{attribute 'GeneratedUsingTerminal: EL6752--0000'}
{attribute addProperty BoxType "EL6752--0000"}
{attribute addProperty Id "InfoDataAT %I*InfoData_90184F0C16"}
{attribute addProperty CRC "554310285"}
{attribute addProperty Size "16"}
TYPE EL6752_210A1A8D EXTENDS EtcSlaveTerminalBase_947E5A46 :
STRUCT
	{attribute addProperty Name "InfoData"}
	InfoData : InfoData_90184F0C;
END_STRUCT
END_TYPE

(* stored: Version 1.2.0.0, ProductVersion 3.1.4024.9
   DUT EL6752_210A1A8D: Id {e3811106-f8e8-4b83-9fd4-58d4e25fdc98} *)
